FUNCTION_BLOCK VAV_SP_CALC (* Calculate Variable Air Volume Controller Set Points *)
  (* Standard: 61499-2 *)
  (* Version 0.0, 2006-05-12, JHC, Holobloc Inc *)
  (* Compiler header: package fb.rt.hvac; *)
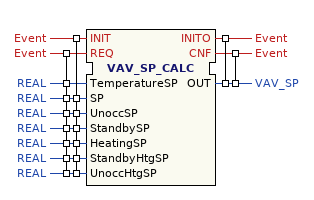
  EVENT_INPUT
    INIT WITH SP, UnoccSP, StandbySP, HeatingSP, StandbyHtgSP, UnoccHtgSP; (* Initialize OUT from SP *)
    REQ WITH TemperatureSP, SP, UnoccSP, StandbySP, HeatingSP, StandbyHtgSP, UnoccHtgSP; (* Compute OUT from TemperatureSP *)
  END_EVENT
  EVENT_OUTPUT
    INITO WITH OUT; (* Confirmation of INIT processing *)
    CNF WITH OUT; (* Confirmation of REQ processing *)
  END_EVENT
  VAR_INPUT
    TemperatureSP : REAL; (* Setpoint from zone controller AI, scaled to same units (eg, deg F) as other inputs *)
    SP : REAL; (* Cooling setpoint. May be modified by the Temperature Setpoint (AI) as an offset *)
    UnoccSP : REAL; (* Unoccupied cooling setpoint.  The offset between SP and UnoccSP will remain the same *)
    StandbySP : REAL; (* Standby cooling setpoint. The offset between SP and StandbySP will remain the same *)
    HeatingSP : REAL; (* Occupied heating setpoint.  The offset between SP and HeatingSP will remain the same *)
    StandbyHtgSP : REAL; (* Standby heating setpoint. The offset between SP and StandbySP will remain the same *)
    UnoccHtgSP : REAL; (* Unoccupied heating setpoint. The offset between SP and UnoccHtgSP will remain the same *)
  END_VAR
  VAR_OUTPUT
    OUT : VAV_SP; (* Computed SP values *)
  END_VAR
  ALGORITHM INIT IN ST: (* Initialize OUT value *)
OUT.SP := SP;
OUT.UnoccSP := UnoccSP;
OUT.StandbySP := StandbySP;
OUT.HeatingSP := HeatingSP;
OUT.UnoccHtgSP := UnoccHtgSP;
OUT.StandbyHtgSP := StandbyHtgSP;
INITO.serviceEvent(this);
  END_ALGORITHM
  ALGORITHM REQ IN ST: (* Set OUT values from TemperatureSP values *)
OUT.SP := TemperatureSP;
OUT.UnoccSP := UnoccSP-SP+TemperatureSP;
OUT.StandbySP := StandbySP-SP+TemperatureSP;
OUT.HeatingSP := HeatingSP-SP+TemperatureSP;
OUT.UnoccHtgSP := UnoccHtgSP-SP+TemperatureSP;
OUT.StandbyHtgSP := StandbyHtgSP-SP+TemperatureSP;
CNF.serviceEvent(this);
  END_ALGORITHM
END_FUNCTION_BLOCK
